// TIA Portal project "TesteFuncional" (V20)

(* hardware
DEVICE "HMI_1"  KTP900 Basic PN
   slot 0: "HMI_1"  KTP900 Basic PN  6AV2 123-2JB03-0AX0  17.0.0.0
   slot 1: "HMI_RT_1"  KTP900 Basic PN  6AV2 123-2JB03-0AX0  17.0.0.0
   slot 5: "HMI_1.IE_CP_1"  PROFINET Interface  17.0.0.0
      slot 1: "PROFINET Interface_1"  PROFINET Interface
         slot 1: "Port_1"  Port
DEVICE "S7-1200 station_1"  S7-1200 Station
   slot 0: "Rack_0"  S7-1200 Rack  Rack  V1.0
   slot 1: "PLC_TesteFuncional"  CPU 1212C DC/DC/DC  6ES7 212-1AE31-0XB0  V3.0
*)

// ===== PLC "PLC_TesteFuncional"  CPU 1212C DC/DC/DC =====

VAR_GLOBAL CONSTANT   // PLC tag table "Default tag table"
   "TIPO_ESTANQUEIDADE" : Int := 1;   // Estanqueidade do sistema de gás (global)
   "TIPO_SEG_ELETRICA" : Int := 2;   // Segurança elétrica: isolamento e fuga (global)
   "TIPO_ELET_SISTEMA" : Int := 3;   // Elétrico do sistema: aterramento, corrente, potência, resistência (global)
   "TIPO_FAISCA" : Int := 4;   // Faísca/ignição: verifica todos os centelhadores (global)
   "TIPO_VAZAO_MAX" : Int := 5;   // Vazão máxima do queimador (por queimador)
   "TIPO_VAZAO_MIN" : Int := 6;   // Vazão mínima com chama mantida (por queimador)
   "TIPO_TEMPERATURA" : Int := 7;   // Temperatura do forno via termopar (por forno)
   "TIPO_ELET_FORNO" : Int := 8;   // Elétrico do elemento do forno (por forno elétrico)
   "TIPO_VISUAL" : Int := 9;   // Inspeção visual do operador (global, no fim)
   "EST_OCIOSO" : Int := 0;   // Aguardando início
   "EST_CONSTRUIR" : Int := 1;   // Montando o plano de execução
   "EST_EXECUTAR" : Int := 2;   // Executando os passos
   "EST_FINALIZADO" : Int := 3;   // Teste concluído, aguardando reset
END_VAR

TYPE "udt_MedicaoFaixa"
   STRUCT
      Nome : String[20];   // Rótulo da medição (ex.: Aterramento)
      Unidade : String[8];   // Unidade de engenharia (ex.: A, Ohm, mbar, °C, L/h)
      LimiteMin : Real;   // Limite inferior; usar -1.0E+09 para desativar
      LimiteMax : Real;   // Limite superior; usar 1.0E+09 para desativar
      ValorNominal : Real;   // Valor central que a simulação busca
      Usado : Bool;   // TRUE se esta sub-medição é avaliada
   END_STRUCT;
END_TYPE

TYPE "udt_DefinicaoPasso"
   STRUCT
      TipoTeste : Int;   // Qual teste (usar as constantes TIPO_)
      Alvo : Int;   // 0 = global; senão índice do queimador/forno
      Descricao : String[40];   // Texto do passo (ex.: Vazao maxima - Queimador 3)
      Duracao : Time;   // Duração do passo
      NumMedicoes : Int;   // Quantidade de sub-medições (1..4)
      Medicoes : Array[1..4] of "udt_MedicaoFaixa";   // Limites/faixas deste passo
   END_STRUCT;
END_TYPE

TYPE "udt_ResultadoPasso"
   STRUCT
      Concluido : Bool;   // TRUE quando o passo terminou
      Aprovado : Bool;   // Resultado: aprovado ou reprovado
      TempoGasto : Time;   // Tempo que o passo levou
      ValoresMedidos : Array[1..4] of Real;   // Valores efetivamente lidos
   END_STRUCT;
END_TYPE

TYPE "udt_Receita"
   STRUCT
      Nome : String[30];   // Nome do modelo (ex.: Fogao A 5Q 2F)
      NumQueimadores : Int;   // Quantidade de queimadores
      NumFornos : Int;   // Quantidade de fornos
      FornoEletrico : Array[1..2] of Bool;   // TRUE = elétrico, FALSE = gás
      HabEstanqueidade : Bool;   // Habilita o teste de estanqueidade
      HabSegEletrica : Bool;   // Habilita o teste de segurança elétrica
      HabEletSistema : Bool;   // Habilita o teste elétrico do sistema
      HabFaisca : Bool;   // Habilita o teste de faísca
      HabVazao : Bool;   // Habilita os testes de vazão
      HabVisual : Bool;   // Habilita a inspeção visual
      DurEstanqueidade : Time;   // Tempo de medição da estanqueidade
      DurSegEletrica : Time;   // Tempo do teste de segurança elétrica
      DurEletSistema : Time;   // Tempo do teste elétrico do sistema
      DurFaisca : Time;   // Tempo do teste de faísca
      DurVazaoMax : Time;   // Tempo da vazão máxima (por queimador)
      DurVazaoMin : Time;   // Tempo da vazão mínima (por queimador)
      DurTemperatura : Time;   // Tempo LIMITE para atingir a faixa
      DurEletForno : Time;   // Tempo do teste elétrico do forno
      Estanqueidade : "udt_MedicaoFaixa";   // Queda de pressão máxima (ΔP)
      SegEletrica : Array[1..2] of "udt_MedicaoFaixa";   // 1=isolamento, 2=corrente de fuga
      EletSistema : Array[1..4] of "udt_MedicaoFaixa";   // 1=aterramento, 2=corrente, 3=potência, 4=resistência
      VazaoMax : Array[1..6] of "udt_MedicaoFaixa";   // Vazão máxima por queimador
      VazaoMin : Array[1..6] of "udt_MedicaoFaixa";   // Vazão mínima por queimador
      Temperatura : Array[1..2] of "udt_MedicaoFaixa";   // Faixa-alvo de temperatura por forno
      EletForno : Array[1..2, 1..3] of "udt_MedicaoFaixa";   // Por forno elétrico: 1=resistência, 2=corrente, 3=potência
   END_STRUCT;
END_TYPE

DATA_BLOCK "DB_Receitas"   // DB1
{ S7_Optimized_Access := 'TRUE' }
VERSION : 0.1
   VAR
      Receitas : Array[1..3] of "udt_Receita";
   END_VAR
BEGIN
   Receitas[2].Nome := 'Fogao B 4Q 1F';
   Receitas[2].NumQueimadores := 4;
   Receitas[2].NumFornos := 1;
   Receitas[2].FornoEletrico[1] := false;
   Receitas[2].FornoEletrico[2] := false;
   Receitas[2].HabEstanqueidade := true;
   Receitas[2].HabSegEletrica := true;
   Receitas[2].HabEletSistema := true;
   Receitas[2].HabFaisca := true;
   Receitas[2].HabVazao := true;
   Receitas[2].HabVisual := true;
   Receitas[2].DurEstanqueidade := T#15s;
   Receitas[2].DurSegEletrica := T#5s;
   Receitas[2].DurEletSistema := T#5s;
   Receitas[2].DurFaisca := T#3s;
   Receitas[2].DurVazaoMax := T#4s;
   Receitas[2].DurVazaoMin := T#4s;
   Receitas[2].DurTemperatura := T#15s;
   Receitas[2].DurEletForno := T#5s;
   Receitas[2].Estanqueidade.Nome := 'Queda Pressao';
   Receitas[2].Estanqueidade.Unidade := 'mbar';
   Receitas[2].Estanqueidade.LimiteMin := -1.0E+09;
   Receitas[2].Estanqueidade.LimiteMax := 1.0;
   Receitas[2].Estanqueidade.ValorNominal := 0.3;
   Receitas[2].Estanqueidade.Usado := true;
   Receitas[2].SegEletrica[1].Nome := 'Isolamento';
   Receitas[2].SegEletrica[1].Unidade := 'MOhm';
   Receitas[2].SegEletrica[1].LimiteMin := 2.0;
   Receitas[2].SegEletrica[1].LimiteMax := 1.0E+09;
   Receitas[2].SegEletrica[1].ValorNominal := 5.0;
   Receitas[2].SegEletrica[1].Usado := true;
   Receitas[2].SegEletrica[2].Nome := 'Corrente Fuga';
   Receitas[2].SegEletrica[2].Unidade := 'mA';
   Receitas[2].SegEletrica[2].LimiteMin := -1.0E+09;
   Receitas[2].SegEletrica[2].LimiteMax := 0.5;
   Receitas[2].SegEletrica[2].ValorNominal := 0.2;
   Receitas[2].SegEletrica[2].Usado := true;
   Receitas[2].EletSistema[1].Nome := 'Aterramento';
   Receitas[2].EletSistema[1].Unidade := 'Ohm';
   Receitas[2].EletSistema[1].LimiteMin := -1.0E+09;
   Receitas[2].EletSistema[1].LimiteMax := 0.1;
   Receitas[2].EletSistema[1].ValorNominal := 0.05;
   Receitas[2].EletSistema[1].Usado := true;
   Receitas[2].EletSistema[2].Usado := true;
   Receitas[2].EletSistema[3].Usado := true;
   Receitas[2].EletSistema[4].Usado := true;
   Receitas[2].EletSistema[2].Nome := 'Corrente';
   Receitas[2].EletSistema[2].Unidade := 'A';
   Receitas[2].EletSistema[2].LimiteMin := 8.0;
   Receitas[2].EletSistema[2].LimiteMax := 12.0;
   Receitas[2].EletSistema[2].ValorNominal := 10.0;
   Receitas[2].EletSistema[3].Nome := 'Potencia';
   Receitas[2].EletSistema[3].Unidade := 'W';
   Receitas[2].EletSistema[3].LimiteMin := 1800.0;
   Receitas[2].EletSistema[3].LimiteMax := 2200.0;
   Receitas[2].EletSistema[3].ValorNominal := 2000.0;
   Receitas[2].EletSistema[4].Nome := 'Resistencia';
   Receitas[2].EletSistema[4].Unidade := 'Ohm';
   Receitas[2].EletSistema[4].LimiteMin := 18.0;
   Receitas[2].EletSistema[4].LimiteMax := 26.0;
   Receitas[2].EletSistema[4].ValorNominal := 22.0;
   Receitas[2].VazaoMax[1].Nome := 'Vazao Max';
   Receitas[2].VazaoMax[1].Unidade := 'L/h';
   Receitas[2].VazaoMax[1].LimiteMin := 180.0;
   Receitas[2].VazaoMax[1].LimiteMax := 240.0;
   Receitas[2].VazaoMax[1].ValorNominal := 210.0;
   Receitas[2].VazaoMax[1].Usado := true;
   Receitas[2].VazaoMax[2].Nome := 'Vazao Max';
   Receitas[2].VazaoMax[2].Unidade := 'L/h';
   Receitas[2].VazaoMax[2].LimiteMin := 180.0;
   Receitas[2].VazaoMax[2].LimiteMax := 240.0;
   Receitas[2].VazaoMax[2].ValorNominal := 210.0;
   Receitas[2].VazaoMax[2].Usado := true;
   Receitas[2].VazaoMax[3].Nome := 'Vazao Max';
   Receitas[2].VazaoMax[3].Unidade := 'L/h';
   Receitas[2].VazaoMax[3].LimiteMin := 180.0;
   Receitas[2].VazaoMax[3].LimiteMax := 240.0;
   Receitas[2].VazaoMax[3].ValorNominal := 210.0;
   Receitas[2].VazaoMax[3].Usado := true;
   Receitas[2].VazaoMax[4].Nome := 'Vazao Max';
   Receitas[2].VazaoMax[4].Unidade := 'L/h';
   Receitas[2].VazaoMax[4].LimiteMin := 180.0;
   Receitas[2].VazaoMax[4].LimiteMax := 240.0;
   Receitas[2].VazaoMax[4].ValorNominal := 210.0;
   Receitas[2].VazaoMax[4].Usado := true;
   Receitas[2].VazaoMax[5].Usado := false;
   Receitas[2].VazaoMax[6].Usado := false;
   Receitas[2].VazaoMin[1].Nome := 'Vazao Min';
   Receitas[2].VazaoMin[1].Unidade := 'L/h';
   Receitas[2].VazaoMin[1].LimiteMin := 25.0;
   Receitas[2].VazaoMin[1].LimiteMax := 55.0;
   Receitas[2].VazaoMin[1].ValorNominal := 40.0;
   Receitas[2].VazaoMin[1].Usado := true;
   Receitas[2].VazaoMin[2].Nome := 'Vazao Min';
   Receitas[2].VazaoMin[2].Unidade := 'L/h';
   Receitas[2].VazaoMin[2].LimiteMin := 25.0;
   Receitas[2].VazaoMin[2].LimiteMax := 55.0;
   Receitas[2].VazaoMin[2].ValorNominal := 40.0;
   Receitas[2].VazaoMin[2].Usado := true;
   Receitas[2].VazaoMin[3].Nome := 'Vazao Min';
   Receitas[2].VazaoMin[3].Unidade := 'L/h';
   Receitas[2].VazaoMin[3].LimiteMin := 25.0;
   Receitas[2].VazaoMin[3].LimiteMax := 55.0;
   Receitas[2].VazaoMin[3].ValorNominal := 40.0;
   Receitas[2].VazaoMin[3].Usado := true;
   Receitas[2].VazaoMin[4].Nome := 'Vazao Min';
   Receitas[2].VazaoMin[4].Unidade := 'L/h';
   Receitas[2].VazaoMin[4].LimiteMin := 25.0;
   Receitas[2].VazaoMin[4].LimiteMax := 55.0;
   Receitas[2].VazaoMin[4].ValorNominal := 40.0;
   Receitas[2].VazaoMin[4].Usado := true;
   Receitas[2].VazaoMin[5].Usado := false;
   Receitas[2].VazaoMin[6].Usado := false;
   Receitas[2].Temperatura[2].Usado := false;
   Receitas[2].Temperatura[1].Nome := 'Temperatura';
   Receitas[2].Temperatura[1].Unidade := '°C';
   Receitas[2].Temperatura[1].LimiteMin := 240.0;
   Receitas[2].Temperatura[1].LimiteMax := 260.0;
   Receitas[2].Temperatura[1].ValorNominal := 250.0;
   Receitas[2].Temperatura[1].Usado := true;
   Receitas[2].EletForno[1,1].Usado := false;
   Receitas[2].EletForno[1,2].Usado := false;
   Receitas[2].EletForno[1,3].Usado := false;
   Receitas[2].EletForno[2,1].Usado := false;
   Receitas[2].EletForno[2,2].Usado := false;
   Receitas[2].EletForno[2,3].Usado := false;
END_DATA_BLOCK

DATA_BLOCK "DB_Execucao"   // DB2
{ S7_Optimized_Access := 'TRUE' }
VERSION : 0.1
   VAR
      ProdutoSelecionado : Int;   // Índice da receita selecionada
      NumeroSerie : Bool;   // Número de série da unidade
      Estado : Int;   // Estado do sequenciador (constantes EST_)
      PassoAtual : Int;   // Passo em execução (1..TotalPassos)
      TotalPassos : Int;   // Total de passos do plano
      TipoTesteAtual : Int;   // Tipo do passo atual (controla a IHM)
      AlvoTextoAtual : String[20];   // Componente sob teste (ex.: Queimador 3)
      NomePassoAtual : String[40];   // Descrição do passo atual
      ValorMedidoAtual : Real;   // Valor principal medido (medidor/barra)
      SubMedidaAtual : Array[1..4] of Real;   // Sub-medições (passos elétricos)
      LimiteMinAtual : Real;   // Limite inferior do passo atual
      LimiteMaxAtual : Real;   // Limite superior do passo atual
      DuracaoPassoAtual : Time;   // Duração total do passo (barra de tempo)
      TempoDecorridoPasso : Time;   // Tempo decorrido do passo (barra de tempo)
      ResultadoPassoAtual : Int;   // 0=rodando, 1=passou, 2=falhou (cor da lâmpada)
      AprovadoGeral : Bool;   // Resultado geral da unidade
      ContadorAprovados : Int;   // Total de unidades aprovadas
      ContadorReprovados : Int;   // Total de unidades reprovadas
      ListaReprovados : String[254];   // Texto dos passos reprovados (retrabalho)
      IniciarTeste : Bool;   // Comando: iniciar teste
      AbortarTeste : Bool;   // Comando: abortar teste
      Resetar : Bool;   // Comando: próxima unidade
      ForcarFalhaPassoAtual : Bool;   // Treino/demo: força a reprovação do passo
      VisualOK : Bool;   // Inspeção visual: aprovado
      VisualNOK : Bool;   // Inspeção visual: reprovado
      PlanoExecucao : Array[1..30] of "udt_DefinicaoPasso";   // Plano de passos montado pelo construtor
      ResultadosPasso : Array[1..30] of "udt_ResultadoPasso";   // Resultado de cada passo executado
   END_VAR
BEGIN
END_DATA_BLOCK

DATA_BLOCK "DB_Simulacao"   // DB3
{ S7_Optimized_Access := 'TRUE' }
VERSION : 0.1
   VAR
      ModeloAtivo : Int := 0;   // Modelo de simulação ativo (= TipoTesteAtual)
      AlvoAtivo : Int := 0;   // Alvo ativo (queimador/forno)
      Habilitar : Bool := false;   // TRUE enquanto a medição corre
      Temperatura : Real := 25.0;   // Temperatura simulada do forno
      TempAmbiente : Real := 25.0;   // Temperatura ambiente
      TempRegime : Real := 0.0;   // Alvo de regime (acima do LimiteMax)
      TauTermico : Real := 0.0;   // Constante de tempo de aquecimento (s)
      TauResfria : Real := 60.0;   // Constante de tempo de resfriamento (s)
      Pressao : Real := 0.0;   // Pressão simulada
      PressaoInicial : Real := 30.0;   // Pressão inicial P0 (mbar)
      DeltaPressao : Real := 0.0;   // Queda de pressão (P0 - atual)
      TaxaVazamento : Real := 0.0;   // Taxa de vazamento (mbar/s)
      Vazao : Real := 0.0;   // Vazão simulada
      ValorEletrico : Array[1..4] of Real;   // Sub-medições elétricas simuladas
      NumCentelhadores : Int := 0;   // Nº de centelhadores (queimadores + fornos a gás)
      FaiscaDetectada : Array[1..8] of Bool;   // Faísca detectada por centelhador
      Semente : DInt := 12345;   // Semente do gerador de ruído (LCG)
      AmplitudeRuido : Real := 0.01;   // Amplitude do ruído (fração do nominal)
   END_VAR
BEGIN
   ValorEletrico[1] := 0.0;
   ValorEletrico[2] := 0.0;
   ValorEletrico[3] := 0.0;
   ValorEletrico[4] := 0.0;
   FaiscaDetectada[1] := false;
   FaiscaDetectada[2] := false;
   FaiscaDetectada[3] := false;
   FaiscaDetectada[4] := false;
   FaiscaDetectada[5] := false;
   FaiscaDetectada[6] := false;
   FaiscaDetectada[7] := false;
   FaiscaDetectada[8] := false;
END_DATA_BLOCK

DATA_BLOCK "DB_iSequenciador"   // DB4
{ S7_Optimized_Access := 'TRUE' }
VERSION : 0.1
// stored: InstanceOfName FB_Sequenciador
"FB_Sequenciador"
BEGIN
END_DATA_BLOCK

FUNCTION_BLOCK "FB_Sequenciador"   // FB1, SCL
{ S7_Optimized_Access := 'TRUE' }
VERSION : 0.1
   VAR
      tmrPasso : TON_TIME;   // Temporizador de espera de cada passo
   END_VAR
   VAR_TEMP
      i : Int;   // Índice de laço
      p : Int;   // Cópia de PassoAtual (índice)
      todosOk : Bool;   // Acumula o "E lógico" dos passos
      ix : Int;
   END_VAR
BEGIN
   // ============================================================
   //  FB_Sequenciador  —  Fase 3
   //  Agora monta o plano real (FC_ConstruirPlano) e mostra os
   //  dados reais do passo. Resultado ainda é forçado (Fase 4 traz
   //  a simulação e a avaliação por faixa).
   // ============================================================

   // ---- Abortar: vale em qualquer estado ----
   IF "DB_Execucao".AbortarTeste THEN
       "DB_Execucao".AbortarTeste := FALSE;
       #tmrPasso(IN := FALSE,
                 PT := T#0s);
       "DB_Execucao".ResultadoPassoAtual := 0;
       "DB_Execucao".Estado := "EST_OCIOSO";
   END_IF;

   CASE "DB_Execucao".Estado OF

       "EST_OCIOSO":
           "DB_Execucao".ResultadoPassoAtual := 0;
           IF "DB_Execucao".IniciarTeste THEN
               "DB_Execucao".IniciarTeste := FALSE;
               FOR #i := 1 TO 30 DO
                   "DB_Execucao".ResultadosPasso[#i].Concluido := FALSE;
                   "DB_Execucao".ResultadosPasso[#i].Aprovado := FALSE;
               END_FOR;
               "DB_Execucao".PassoAtual := 0;
               "DB_Execucao".AprovadoGeral := FALSE;
               "DB_Execucao".Estado := "EST_CONSTRUIR";
           END_IF;

       "EST_CONSTRUIR":
           #ix := "DB_Execucao".ProdutoSelecionado;
           IF (#ix < 1) OR (#ix > 3) THEN
               #ix := 2;                       // proteção: Fogão B por padrão
           END_IF;
           // monta o plano a partir da receita selecionada
           "FC_ConstruirPlano"(receita := "DB_Receitas".Receitas[#ix],
                               plano := "DB_Execucao".PlanoExecucao,
                               totalPassos => "DB_Execucao".TotalPassos);
           "DB_Execucao".PassoAtual := 1;
           "DB_Execucao".Estado := "EST_EXECUTAR";

       "EST_EXECUTAR":
           #p := "DB_Execucao".PassoAtual;

           // ----- espelho do passo atual (para a IHM) -----
           "DB_Execucao".TipoTesteAtual := "DB_Execucao".PlanoExecucao[#p].TipoTeste;
           "DB_Execucao".NomePassoAtual := "DB_Execucao".PlanoExecucao[#p].Descricao;
           "DB_Execucao".DuracaoPassoAtual := "DB_Execucao".PlanoExecucao[#p].Duracao;

           // texto do alvo (Sistema / Queimador N / Forno N)
           IF "DB_Execucao".PlanoExecucao[#p].Alvo = 0 THEN
               "DB_Execucao".AlvoTextoAtual := 'Sistema';
           ELSIF ("DB_Execucao".TipoTesteAtual = "TIPO_VAZAO_MAX")
               OR ("DB_Execucao".TipoTesteAtual = "TIPO_VAZAO_MIN") THEN
               "DB_Execucao".AlvoTextoAtual := CONCAT(IN1 := 'Queimador ',
                                                      IN2 := INT_TO_STRING("DB_Execucao".PlanoExecucao[#p].Alvo));
           ELSE
               "DB_Execucao".AlvoTextoAtual := CONCAT(IN1 := 'Forno ',
                                                      IN2 := INT_TO_STRING("DB_Execucao".PlanoExecucao[#p].Alvo));
           END_IF;

           // limites principais (1ª medição) p/ exibição
           IF "DB_Execucao".PlanoExecucao[#p].NumMedicoes >= 1 THEN
               "DB_Execucao".LimiteMinAtual := "DB_Execucao".PlanoExecucao[#p].Medicoes[1].LimiteMin;
               "DB_Execucao".LimiteMaxAtual := "DB_Execucao".PlanoExecucao[#p].Medicoes[1].LimiteMax;
           ELSE
               "DB_Execucao".LimiteMinAtual := 0.0;
               "DB_Execucao".LimiteMaxAtual := 0.0;
           END_IF;

           "DB_Execucao".ResultadoPassoAtual := 0;     // rodando

           // espera a DURAÇÃO REAL do passo
           #tmrPasso(IN := TRUE,
                     PT := "DB_Execucao".PlanoExecucao[#p].Duracao);
           "DB_Execucao".TempoDecorridoPasso := #tmrPasso.ET;

           IF #tmrPasso.Q THEN
               // ----- força APROVADO (ainda sem simulação) -----
               "DB_Execucao".ResultadosPasso[#p].Concluido := TRUE;
               "DB_Execucao".ResultadosPasso[#p].Aprovado := TRUE;
               "DB_Execucao".ResultadosPasso[#p].TempoGasto := #tmrPasso.ET;
               "DB_Execucao".ResultadoPassoAtual := 1;

               #tmrPasso(IN := FALSE,
                         PT := T#0s);

               IF #p < "DB_Execucao".TotalPassos THEN
                   "DB_Execucao".PassoAtual := #p + 1;
               ELSE
                   #todosOk := TRUE;
                   FOR #i := 1 TO "DB_Execucao".TotalPassos DO
                       IF NOT "DB_Execucao".ResultadosPasso[#i].Aprovado THEN
                           #todosOk := FALSE;
                       END_IF;
                   END_FOR;
                   "DB_Execucao".AprovadoGeral := #todosOk;
                   IF #todosOk THEN
                       "DB_Execucao".ContadorAprovados := "DB_Execucao".ContadorAprovados + 1;
                   ELSE
                       "DB_Execucao".ContadorReprovados := "DB_Execucao".ContadorReprovados + 1;
                   END_IF;
                   "DB_Execucao".Estado := "EST_FINALIZADO";
               END_IF;
           END_IF;

       "EST_FINALIZADO":
           IF "DB_Execucao".Resetar THEN
               "DB_Execucao".Resetar := FALSE;
               "DB_Execucao".Estado := "EST_OCIOSO";
           END_IF;

   END_CASE;
END_FUNCTION_BLOCK

FUNCTION "FC_ConstruirPlano" : Void   // FC1, SCL
{ S7_Optimized_Access := 'TRUE' }
VERSION : 0.1
   VAR_OUTPUT
      totalPassos : Int;   // Quantidade de passos gerados
   END_VAR
   VAR_IN_OUT
      receita : "udt_Receita";   // Receita selecionada (somente leitura aqui)
      plano : Array[1..30] of "udt_DefinicaoPasso";   // Plano a ser preenchido
   END_VAR
   VAR_TEMP
      idx : Int;   // Índice do passo sendo gravado
      i : Int;   // Laço dos queimadores
      j : Int;   // Laço dos fornos
   END_VAR
BEGIN
   // ============================================================
   //  FC_ConstruirPlano  —  Fase 3
   //  Expande a receita em uma lista de passos (PlanoExecucao),
   //  na ordem fixa de segurança. Retorna o total em totalPassos.
   // ============================================================

   #idx := 0;

   // ---------- 1) Testes globais, na ordem de segurança ----------
   IF #receita.HabEstanqueidade THEN
       #idx := #idx + 1;
       #plano[#idx].TipoTeste := "TIPO_ESTANQUEIDADE";
       #plano[#idx].Alvo := 0;
       #plano[#idx].Duracao := #receita.DurEstanqueidade;
       #plano[#idx].NumMedicoes := 1;
       #plano[#idx].Medicoes[1] := #receita.Estanqueidade;
       #plano[#idx].Descricao := 'Estanqueidade';
   END_IF;

   IF #receita.HabSegEletrica THEN
       #idx := #idx + 1;
       #plano[#idx].TipoTeste := "TIPO_SEG_ELETRICA";
       #plano[#idx].Alvo := 0;
       #plano[#idx].Duracao := #receita.DurSegEletrica;
       #plano[#idx].NumMedicoes := 2;
       #plano[#idx].Medicoes[1] := #receita.SegEletrica[1];
       #plano[#idx].Medicoes[2] := #receita.SegEletrica[2];
       #plano[#idx].Descricao := 'Seguranca eletrica';
   END_IF;

   IF #receita.HabEletSistema THEN
       #idx := #idx + 1;
       #plano[#idx].TipoTeste := "TIPO_ELET_SISTEMA";
       #plano[#idx].Alvo := 0;
       #plano[#idx].Duracao := #receita.DurEletSistema;
       #plano[#idx].NumMedicoes := 4;
       #plano[#idx].Medicoes[1] := #receita.EletSistema[1];
       #plano[#idx].Medicoes[2] := #receita.EletSistema[2];
       #plano[#idx].Medicoes[3] := #receita.EletSistema[3];
       #plano[#idx].Medicoes[4] := #receita.EletSistema[4];
       #plano[#idx].Descricao := 'Eletrico do sistema';
   END_IF;

   IF #receita.HabFaisca THEN
       #idx := #idx + 1;
       #plano[#idx].TipoTeste := "TIPO_FAISCA";
       #plano[#idx].Alvo := 0;
       #plano[#idx].Duracao := #receita.DurFaisca;
       #plano[#idx].NumMedicoes := 0;          // faísca não tem faixa numérica
       #plano[#idx].Descricao := 'Faisca - todos';
   END_IF;

   // ---------- 2) Queimadores: Vazão máx -> Vazão mín ----------
   IF #receita.HabVazao THEN
       FOR #i := 1 TO #receita.NumQueimadores DO
           // Vazão máxima
           #idx := #idx + 1;
           #plano[#idx].TipoTeste := "TIPO_VAZAO_MAX";
           #plano[#idx].Alvo := #i;
           #plano[#idx].Duracao := #receita.DurVazaoMax;
           #plano[#idx].NumMedicoes := 1;
           #plano[#idx].Medicoes[1] := #receita.VazaoMax[#i];
           #plano[#idx].Descricao := CONCAT(IN1 := 'Vazao maxima - Queimador ',
                                            IN2 := INT_TO_STRING(#i));
           // Vazão mínima
           #idx := #idx + 1;
           #plano[#idx].TipoTeste := "TIPO_VAZAO_MIN";
           #plano[#idx].Alvo := #i;
           #plano[#idx].Duracao := #receita.DurVazaoMin;
           #plano[#idx].NumMedicoes := 1;
           #plano[#idx].Medicoes[1] := #receita.VazaoMin[#i];
           #plano[#idx].Descricao := CONCAT(IN1 := 'Vazao minima - Queimador ',
                                            IN2 := INT_TO_STRING(#i));
       END_FOR;
   END_IF;

   // ---------- 3) Fornos: Temperatura (+ Elétrico se for elétrico) ----------
   FOR #j := 1 TO #receita.NumFornos DO
       // Temperatura
       #idx := #idx + 1;
       #plano[#idx].TipoTeste := "TIPO_TEMPERATURA";
       #plano[#idx].Alvo := #j;
       #plano[#idx].Duracao := #receita.DurTemperatura;
       #plano[#idx].NumMedicoes := 1;
       #plano[#idx].Medicoes[1] := #receita.Temperatura[#j];
       #plano[#idx].Descricao := CONCAT(IN1 := 'Temperatura - Forno ',
                                        IN2 := INT_TO_STRING(#j));
       // Elétrico do elemento — só se o forno for elétrico
       IF #receita.FornoEletrico[#j] THEN
           #idx := #idx + 1;
           #plano[#idx].TipoTeste := "TIPO_ELET_FORNO";
           #plano[#idx].Alvo := #j;
           #plano[#idx].Duracao := #receita.DurEletForno;
           #plano[#idx].NumMedicoes := 3;
           #plano[#idx].Medicoes[1] := #receita.EletForno[#j, 1];
           #plano[#idx].Medicoes[2] := #receita.EletForno[#j, 2];
           #plano[#idx].Medicoes[3] := #receita.EletForno[#j, 3];
           #plano[#idx].Descricao := CONCAT(IN1 := 'Eletrico do elemento - Forno ',
                                            IN2 := INT_TO_STRING(#j));
       END_IF;
   END_FOR;

   // ---------- 4) Inspeção visual no fim ----------
   IF #receita.HabVisual THEN
       #idx := #idx + 1;
       #plano[#idx].TipoTeste := "TIPO_VISUAL";
       #plano[#idx].Alvo := 0;
       #plano[#idx].Duracao := T#0s;       // espera o operador (Fase 5)
       #plano[#idx].NumMedicoes := 0;
       #plano[#idx].Descricao := 'Inspecao visual';
   END_IF;

   #totalPassos := #idx;
END_FUNCTION

ORGANIZATION_BLOCK "Main"   // OB1, LAD, ProgramCycle
TITLE = "Main Program Sweep (Cycle)"
{ S7_Optimized_Access := 'TRUE' }
VERSION : 0.1
BEGIN

REGION Network 1
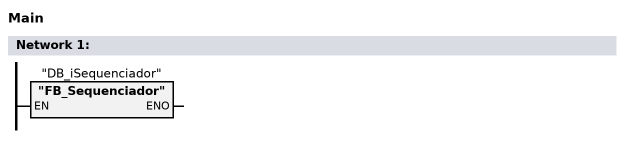
   RUNG wire#powerrail
      "DB_iSequenciador"()
   END_RUNG
   // the same network as SCL:
   "DB_iSequenciador"();   // "FB_Sequenciador"
END_REGION
END_ORGANIZATION_BLOCK

(* ===== HMI "HMI_RT_1" =====

screen "Root screen" 800x480, template "Template_1"
   TextField "HmiScreenItemData" at 80,226 size 640x22; Text 'Welcome to HMI_1 (KTP900 Basic+ PN)!'
*)